# EPICS StreamDevice protocol: DG645Sup/DG645.proto
Terminator = CR LF;

getIDN {
    out "*IDN?";
    in "%\$1[^\n]";
    ExtraInput = Ignore;
}

# Generic

cmd {
    out "\$1";
}

setD {
    out "\$1 %d";
}

getD {
    out "\$1?";
    in "%d";
    ExtraInput = Ignore;
}

getWF {
    out "\$2";
    in "%\$1[^\r\n]";
}

# Status and display command

# Trigger

# Delay

delay {
    out "DLAY %(\$1ChannelEdge)d,%(\$1ChannelLink)d,%e";
}
